FUNCTION_BLOCK FB_Reactor_Set_Ext_FAT EXTENDS FB_Reactor_Set
VAR_INPUT
END_VAR
VAR_OUTPUT
END_VAR
VAR
	fb_ReadJsonFAT : FB_ReadWrite_Json;
	sita_bit1 : BOOL;
END_VAR

fb_ReadJsonFAT(
		i_ExecuteRead := sita_bit1,
		i_Json_FilePath := FAT.json_file_path,
		i_JsonStructure := 'FAT.st_steam_desorption');

//Steam_Desorption_FAT();	

SUPER^();

END_FUNCTION_BLOCK

(* stored: Version 1.1.0.1, ProductVersion 3.1.4024.12
   POU FB_Reactor_Set_Ext_FAT: Id {df9eef0f-6051-440c-9027-049bdb3cca1d}, SpecialFunc None *)
